// TIA Portal V16 export
// export: Created 2021-12-01T20:36:14.8298503Z, ExportSetting WithDefaults, DisplayName Totally Integrated Automation Portal, DisplayVersion V16 Update 4, DisplayName TIA Portal Version Control Interface, DisplayVersion V16 Update 2, DisplayName TIA Portal Openness, DisplayVersion V16 Update 4, DisplayName SINAMICS Startdrive Advanced, DisplayVersion V16 Update 5, DisplayName SINAMICS Startdrive G130, G150, S120, S150, SINAMICS MV, S210, DisplayVersion V16 Update 5, DisplayName SINAMICS Startdrive G110M, G120, G120C, G120D, G120P, G115D, DisplayVersion V16 Update 5, DisplayName STEP 7 Professional, DisplayVersion V16 Update 4, DisplayName STEP 7 Safety, DisplayVersion V16, DisplayName WinCC Advanced, DisplayVersion V16 Update 4
FUNCTION "ST00320_FC" : Void   // FC165, LAD
TITLE = ST00320
{ S7_Optimized_Access := 'TRUE' }
VERSION : 0.1
// stored: AutoNumber true, IsIECCheckEnabled false, SetENOAutomatically false, UDAEnableTagReadback false
   VAR_IN_OUT
      OPMODE : "OPMODE_OUT_UDT";
      HMI_EXTENSION : "HMI_EXTENSION_PANEL_UDT";
   END_VAR
   VAR_TEMP
      EmptyHS : "RT_HANDSHAKE_UDT";
   END_VAR
BEGIN

REGION Network 1: Move Opmode
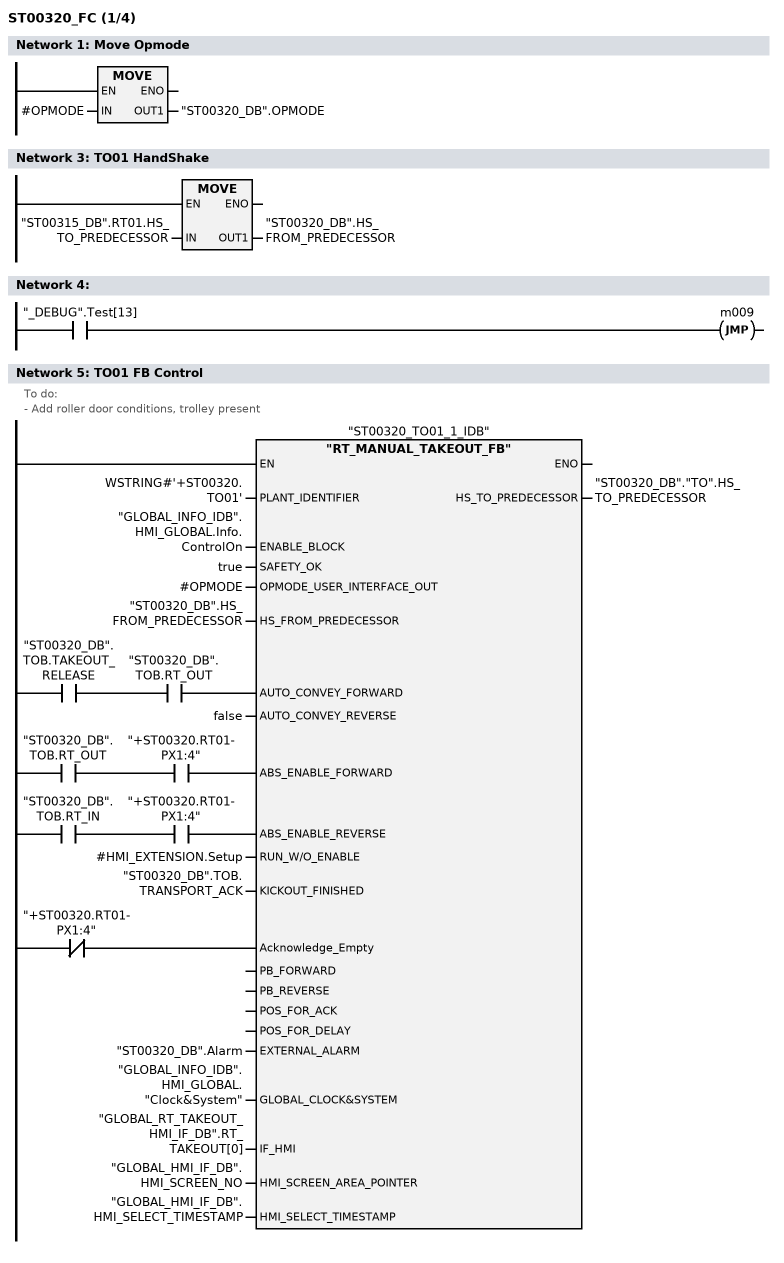
   RUNG wire#powerrail
      Move(in := #OPMODE, out1 => "ST00320_DB".OPMODE)
   END_RUNG
   // the same network as SCL:
   "ST00320_DB".OPMODE := #OPMODE;
END_REGION

REGION Network 2: *******************TO01 Control*******************
END_REGION

REGION Network 3: TO01 HandShake
   RUNG wire#powerrail
      Move(in := "ST00315_DB".RT01.HS_TO_PREDECESSOR, out1 => "ST00320_DB".HS_FROM_PREDECESSOR)
   END_RUNG
   // the same network as SCL:
   "ST00320_DB".HS_FROM_PREDECESSOR := "ST00315_DB".RT01.HS_TO_PREDECESSOR;
END_REGION

REGION Network 4
   RUNG wire#powerrail
      Contact( "_DEBUG".Test[13] )
      JumpCoil( m009 )
   END_RUNG
   // the same network as SCL:
   IF "_DEBUG".Test[13] THEN GOTO m009; END_IF;
END_REGION

REGION Network 5: TO01 FB Control
   // To do:
   // - Add roller door conditions, trolley present
   RUNG wire#powerrail
      "ST00320_TO01_1_IDB"(AUTO_CONVEY_FORWARD := wire#w1, ABS_ENABLE_FORWARD := wire#w2, ABS_ENABLE_REVERSE := wire#w3, Acknowledge_Empty := wire#w4, PLANT_IDENTIFIER := WSTRING#'+ST00320.TO01', ENABLE_BLOCK := "GLOBAL_INFO_IDB".HMI_GLOBAL.Info.ControlOn, SAFETY_OK := true, OPMODE_USER_INTERFACE_OUT := #OPMODE, HS_FROM_PREDECESSOR := "ST00320_DB".HS_FROM_PREDECESSOR, AUTO_CONVEY_REVERSE := false, "RUN_W/O_ENABLE" := #HMI_EXTENSION.Setup, KICKOUT_FINISHED := "ST00320_DB".TOB.TRANSPORT_ACK, PB_FORWARD :=, PB_REVERSE :=, POS_FOR_ACK :=, POS_FOR_DELAY :=, EXTERNAL_ALARM := "ST00320_DB".Alarm, "GLOBAL_CLOCK&SYSTEM" := "GLOBAL_INFO_IDB".HMI_GLOBAL."Clock&System", IF_HMI := "GLOBAL_RT_TAKEOUT_HMI_IF_DB".RT_TAKEOUT[0], HMI_SCREEN_AREA_POINTER := "GLOBAL_HMI_IF_DB".HMI_SCREEN_NO, HMI_SELECT_TIMESTAMP := "GLOBAL_HMI_IF_DB".HMI_SELECT_TIMESTAMP, HS_TO_PREDECESSOR => "ST00320_DB"."TO".HS_TO_PREDECESSOR)
   END_RUNG
   RUNG wire#powerrail
      Contact( "ST00320_DB".TOB.TAKEOUT_RELEASE )
      Contact( "ST00320_DB".TOB.RT_OUT )
   END_RUNG wire#w1
   RUNG wire#powerrail
      Contact( "ST00320_DB".TOB.RT_OUT )
      Contact( "+ST00320.RT01-PX1:4" )
   END_RUNG wire#w2
   RUNG wire#powerrail
      Contact( "ST00320_DB".TOB.RT_IN )
      Contact( "+ST00320.RT01-PX1:4" )
   END_RUNG wire#w3
   RUNG wire#powerrail
      I_Contact( "+ST00320.RT01-PX1:4" )
   END_RUNG wire#w4
   // the same network as SCL:
   "ST00320_TO01_1_IDB"(PLANT_IDENTIFIER := WSTRING#'+ST00320.TO01',   // "RT_MANUAL_TAKEOUT_FB"
                        ENABLE_BLOCK := "GLOBAL_INFO_IDB".HMI_GLOBAL.Info.ControlOn,
                        SAFETY_OK := true,
                        OPMODE_USER_INTERFACE_OUT := #OPMODE,
                        HS_FROM_PREDECESSOR := "ST00320_DB".HS_FROM_PREDECESSOR,
                        AUTO_CONVEY_FORWARD := "ST00320_DB".TOB.TAKEOUT_RELEASE AND "ST00320_DB".TOB.RT_OUT,
                        AUTO_CONVEY_REVERSE := false,
                        ABS_ENABLE_FORWARD := "ST00320_DB".TOB.RT_OUT AND "+ST00320.RT01-PX1:4",
                        ABS_ENABLE_REVERSE := "ST00320_DB".TOB.RT_IN AND "+ST00320.RT01-PX1:4",
                        "RUN_W/O_ENABLE" := #HMI_EXTENSION.Setup,
                        KICKOUT_FINISHED := "ST00320_DB".TOB.TRANSPORT_ACK,
                        Acknowledge_Empty := NOT "+ST00320.RT01-PX1:4",
                        EXTERNAL_ALARM := "ST00320_DB".Alarm,
                        "GLOBAL_CLOCK&SYSTEM" := "GLOBAL_INFO_IDB".HMI_GLOBAL."Clock&System",
                        IF_HMI := "GLOBAL_RT_TAKEOUT_HMI_IF_DB".RT_TAKEOUT[0],
                        HMI_SCREEN_AREA_POINTER := "GLOBAL_HMI_IF_DB".HMI_SCREEN_NO,
                        HMI_SELECT_TIMESTAMP := "GLOBAL_HMI_IF_DB".HMI_SELECT_TIMESTAMP,
                        HS_TO_PREDECESSOR => "ST00320_DB"."TO".HS_TO_PREDECESSOR);
END_REGION

REGION Network 6: Takeout Box
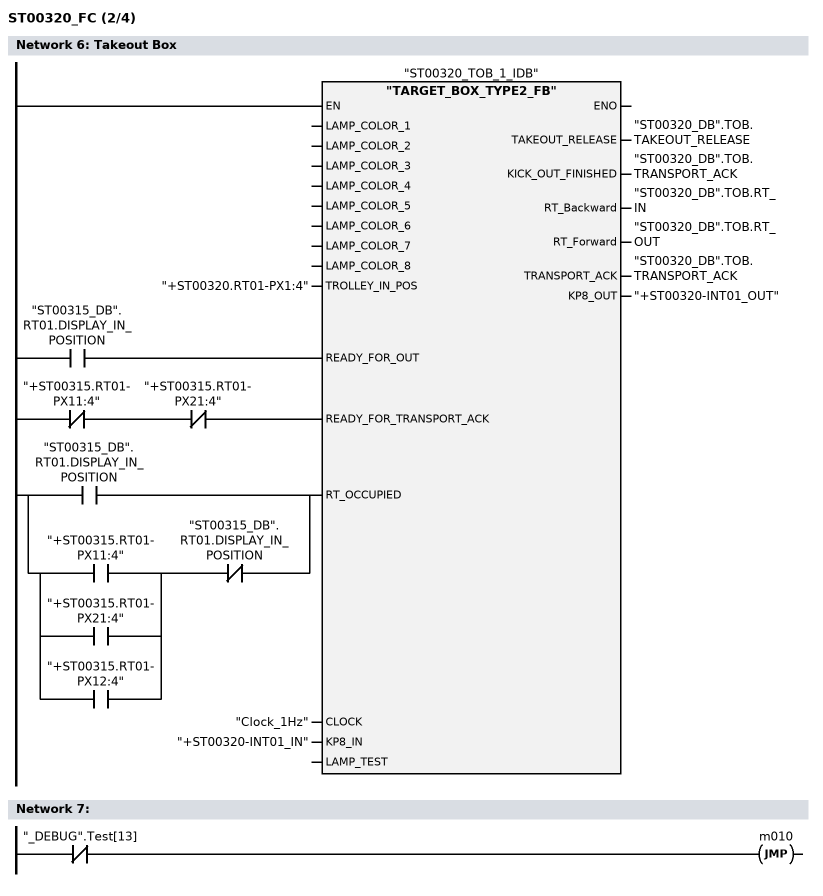
   RUNG wire#powerrail
      "ST00320_TOB_1_IDB"(READY_FOR_OUT := wire#w1, READY_FOR_TRANSPORT_ACK := wire#w2, RT_OCCUPIED := wire#w4, LAMP_COLOR_1 :=, LAMP_COLOR_2 :=, LAMP_COLOR_3 :=, LAMP_COLOR_4 :=, LAMP_COLOR_5 :=, LAMP_COLOR_6 :=, LAMP_COLOR_7 :=, LAMP_COLOR_8 :=, TROLLEY_IN_POS := "+ST00320.RT01-PX1:4", CLOCK := "Clock_1Hz", KP8_IN := "+ST00320-INT01_IN", LAMP_TEST :=, TAKEOUT_RELEASE => "ST00320_DB".TOB.TAKEOUT_RELEASE, KICK_OUT_FINISHED => "ST00320_DB".TOB.TRANSPORT_ACK, RT_Backward => "ST00320_DB".TOB.RT_IN, RT_Forward => "ST00320_DB".TOB.RT_OUT, TRANSPORT_ACK => "ST00320_DB".TOB.TRANSPORT_ACK, KP8_OUT => "+ST00320-INT01_OUT")
   END_RUNG
   RUNG wire#powerrail
      Contact( "ST00315_DB".RT01.DISPLAY_IN_POSITION )
   END_RUNG wire#w1
   RUNG wire#powerrail
      I_Contact( "+ST00315.RT01-PX11:4" )
      I_Contact( "+ST00315.RT01-PX21:4" )
   END_RUNG wire#w2
   RUNG wire#powerrail
      Contact( "ST00315_DB".RT01.DISPLAY_IN_POSITION )
   END_RUNG wire#w4
   RUNG wire#powerrail
      Contact( "+ST00315.RT01-PX11:4" )
      wire#w3
      I_Contact( "ST00315_DB".RT01.DISPLAY_IN_POSITION )
   END_RUNG wire#w4
   RUNG wire#powerrail
      Contact( "+ST00315.RT01-PX21:4" )
   END_RUNG wire#w3
   RUNG wire#powerrail
      Contact( "+ST00315.RT01-PX12:4" )
   END_RUNG wire#w3
   // the same network as SCL:
   "ST00320_TOB_1_IDB"(TROLLEY_IN_POS := "+ST00320.RT01-PX1:4",   // "TARGET_BOX_TYPE2_FB"
                       READY_FOR_OUT := "ST00315_DB".RT01.DISPLAY_IN_POSITION,
                       READY_FOR_TRANSPORT_ACK := NOT "+ST00315.RT01-PX11:4" AND NOT "+ST00315.RT01-PX21:4",
                       RT_OCCUPIED := "ST00315_DB".RT01.DISPLAY_IN_POSITION OR (("+ST00315.RT01-PX11:4" OR "+ST00315.RT01-PX21:4" OR "+ST00315.RT01-PX12:4") AND NOT "ST00315_DB".RT01.DISPLAY_IN_POSITION),
                       CLOCK := "Clock_1Hz",
                       KP8_IN := "+ST00320-INT01_IN",
                       TAKEOUT_RELEASE => "ST00320_DB".TOB.TAKEOUT_RELEASE,
                       KICK_OUT_FINISHED => "ST00320_DB".TOB.TRANSPORT_ACK,
                       RT_Backward => "ST00320_DB".TOB.RT_IN,
                       RT_Forward => "ST00320_DB".TOB.RT_OUT,
                       TRANSPORT_ACK => "ST00320_DB".TOB.TRANSPORT_ACK,
                       KP8_OUT => "+ST00320-INT01_OUT");
END_REGION

REGION Network 7
   RUNG wire#powerrail
      I_Contact( "_DEBUG".Test[13] )
      JumpCoil( m010 )
   END_RUNG
   // the same network as SCL:
   IF NOT "_DEBUG".Test[13] THEN GOTO m010; END_IF;
END_REGION

REGION Network 8: ----test----TO01 HandShake
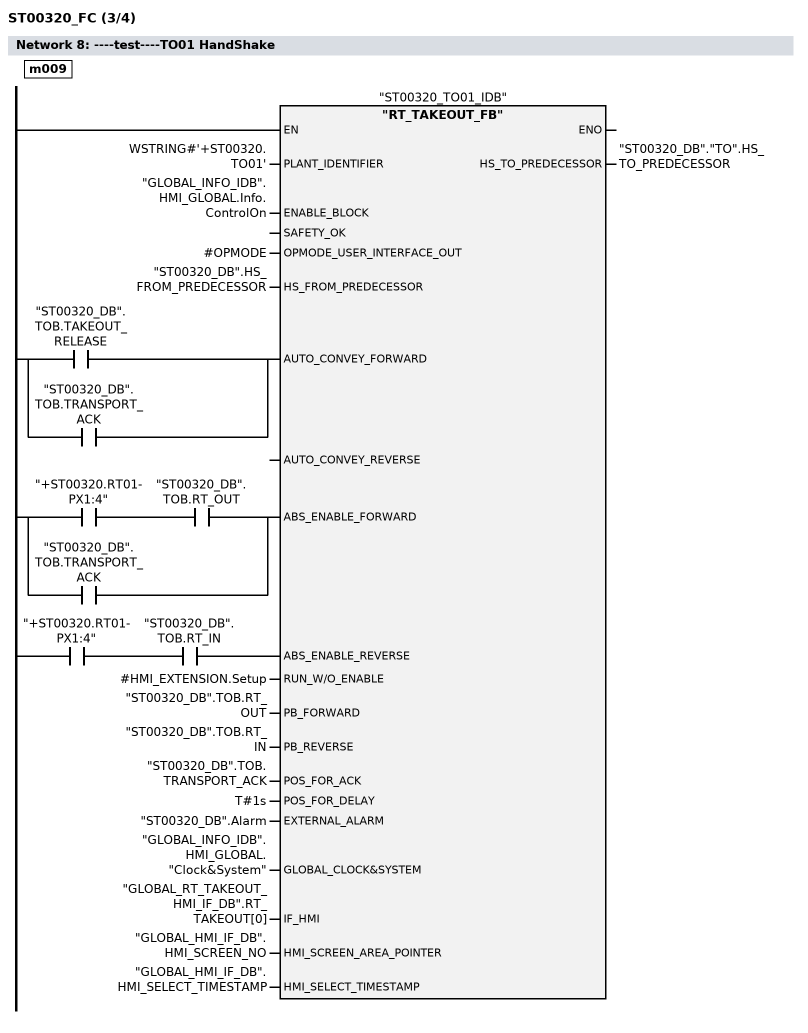
   Label( m009 )
   RUNG wire#powerrail
      "ST00320_TO01_IDB"(AUTO_CONVEY_FORWARD := wire#w1, ABS_ENABLE_FORWARD := wire#w2, ABS_ENABLE_REVERSE := wire#w3, PLANT_IDENTIFIER := WSTRING#'+ST00320.TO01', ENABLE_BLOCK := "GLOBAL_INFO_IDB".HMI_GLOBAL.Info.ControlOn, SAFETY_OK :=, OPMODE_USER_INTERFACE_OUT := #OPMODE, HS_FROM_PREDECESSOR := "ST00320_DB".HS_FROM_PREDECESSOR, AUTO_CONVEY_REVERSE :=, "RUN_W/O_ENABLE" := #HMI_EXTENSION.Setup, PB_FORWARD := "ST00320_DB".TOB.RT_OUT, PB_REVERSE := "ST00320_DB".TOB.RT_IN, POS_FOR_ACK := "ST00320_DB".TOB.TRANSPORT_ACK, POS_FOR_DELAY := T#1s, EXTERNAL_ALARM := "ST00320_DB".Alarm, "GLOBAL_CLOCK&SYSTEM" := "GLOBAL_INFO_IDB".HMI_GLOBAL."Clock&System", IF_HMI := "GLOBAL_RT_TAKEOUT_HMI_IF_DB".RT_TAKEOUT[0], HMI_SCREEN_AREA_POINTER := "GLOBAL_HMI_IF_DB".HMI_SCREEN_NO, HMI_SELECT_TIMESTAMP := "GLOBAL_HMI_IF_DB".HMI_SELECT_TIMESTAMP, HS_TO_PREDECESSOR => "ST00320_DB"."TO".HS_TO_PREDECESSOR)
   END_RUNG
   RUNG wire#powerrail
      Contact( "ST00320_DB".TOB.TAKEOUT_RELEASE )
   END_RUNG wire#w1
   RUNG wire#powerrail
      Contact( "ST00320_DB".TOB.TRANSPORT_ACK )
   END_RUNG wire#w1
   RUNG wire#powerrail
      Contact( "+ST00320.RT01-PX1:4" )
      Contact( "ST00320_DB".TOB.RT_OUT )
   END_RUNG wire#w2
   RUNG wire#powerrail
      Contact( "ST00320_DB".TOB.TRANSPORT_ACK )
   END_RUNG wire#w2
   RUNG wire#powerrail
      Contact( "+ST00320.RT01-PX1:4" )
      Contact( "ST00320_DB".TOB.RT_IN )
   END_RUNG wire#w3
   // the same network as SCL:
   m009:
   "ST00320_TO01_IDB"(PLANT_IDENTIFIER := WSTRING#'+ST00320.TO01',   // "RT_TAKEOUT_FB"
                      ENABLE_BLOCK := "GLOBAL_INFO_IDB".HMI_GLOBAL.Info.ControlOn,
                      OPMODE_USER_INTERFACE_OUT := #OPMODE,
                      HS_FROM_PREDECESSOR := "ST00320_DB".HS_FROM_PREDECESSOR,
                      AUTO_CONVEY_FORWARD := "ST00320_DB".TOB.TAKEOUT_RELEASE OR "ST00320_DB".TOB.TRANSPORT_ACK,
                      ABS_ENABLE_FORWARD := ("+ST00320.RT01-PX1:4" AND "ST00320_DB".TOB.RT_OUT) OR "ST00320_DB".TOB.TRANSPORT_ACK,
                      ABS_ENABLE_REVERSE := "+ST00320.RT01-PX1:4" AND "ST00320_DB".TOB.RT_IN,
                      "RUN_W/O_ENABLE" := #HMI_EXTENSION.Setup,
                      PB_FORWARD := "ST00320_DB".TOB.RT_OUT,
                      PB_REVERSE := "ST00320_DB".TOB.RT_IN,
                      POS_FOR_ACK := "ST00320_DB".TOB.TRANSPORT_ACK,
                      POS_FOR_DELAY := T#1s,
                      EXTERNAL_ALARM := "ST00320_DB".Alarm,
                      "GLOBAL_CLOCK&SYSTEM" := "GLOBAL_INFO_IDB".HMI_GLOBAL."Clock&System",
                      IF_HMI := "GLOBAL_RT_TAKEOUT_HMI_IF_DB".RT_TAKEOUT[0],
                      HMI_SCREEN_AREA_POINTER := "GLOBAL_HMI_IF_DB".HMI_SCREEN_NO,
                      HMI_SELECT_TIMESTAMP := "GLOBAL_HMI_IF_DB".HMI_SELECT_TIMESTAMP,
                      HS_TO_PREDECESSOR => "ST00320_DB"."TO".HS_TO_PREDECESSOR);
END_REGION

REGION Network 9: Takeout Box Standar
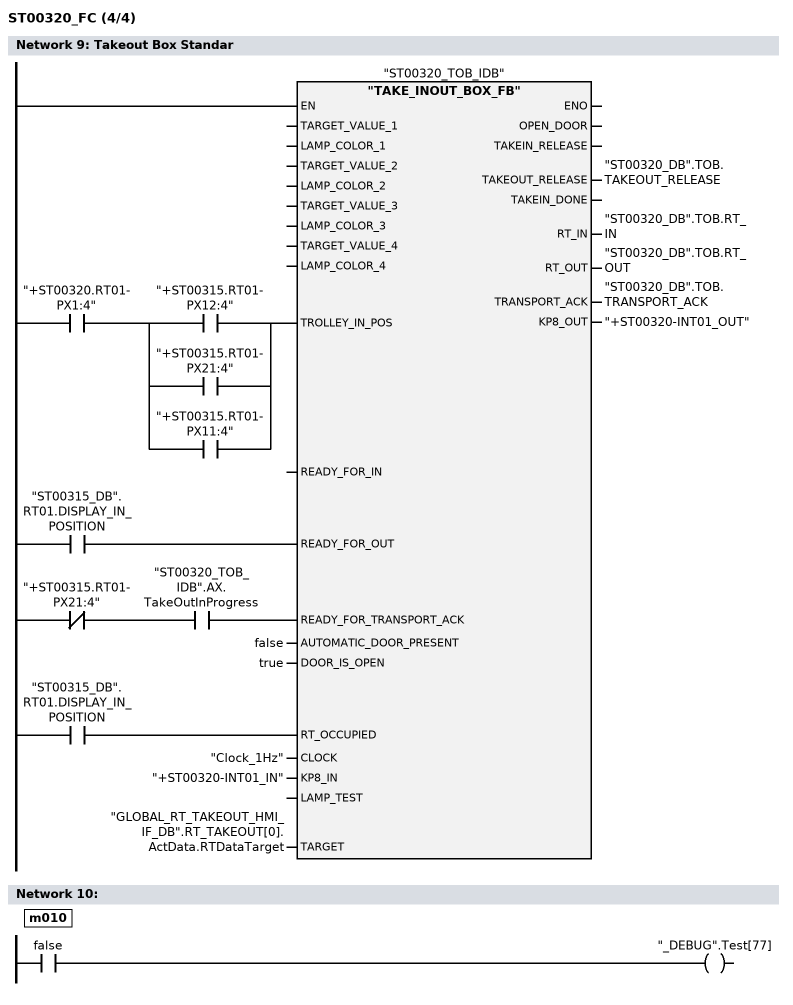
   RUNG wire#powerrail
      "ST00320_TOB_IDB"(TROLLEY_IN_POS := wire#w2, READY_FOR_OUT := wire#w3, READY_FOR_TRANSPORT_ACK := wire#w4, RT_OCCUPIED := wire#w5, TARGET_VALUE_1 :=, LAMP_COLOR_1 :=, TARGET_VALUE_2 :=, LAMP_COLOR_2 :=, TARGET_VALUE_3 :=, LAMP_COLOR_3 :=, TARGET_VALUE_4 :=, LAMP_COLOR_4 :=, READY_FOR_IN :=, AUTOMATIC_DOOR_PRESENT := false, DOOR_IS_OPEN := true, CLOCK := "Clock_1Hz", KP8_IN := "+ST00320-INT01_IN", LAMP_TEST :=, TARGET := "GLOBAL_RT_TAKEOUT_HMI_IF_DB".RT_TAKEOUT[0].ActData.RTDataTarget, OPEN_DOOR =>, TAKEIN_RELEASE =>, TAKEOUT_RELEASE => "ST00320_DB".TOB.TAKEOUT_RELEASE, TAKEIN_DONE =>, RT_IN => "ST00320_DB".TOB.RT_IN, RT_OUT => "ST00320_DB".TOB.RT_OUT, TRANSPORT_ACK => "ST00320_DB".TOB.TRANSPORT_ACK, KP8_OUT => "+ST00320-INT01_OUT")
   END_RUNG
   RUNG wire#powerrail
      Contact( "+ST00320.RT01-PX1:4" )
      wire#w1
      Contact( "+ST00315.RT01-PX12:4" )
   END_RUNG wire#w2
   RUNG wire#w1
      Contact( "+ST00315.RT01-PX21:4" )
   END_RUNG wire#w2
   RUNG wire#w1
      Contact( "+ST00315.RT01-PX11:4" )
   END_RUNG wire#w2
   RUNG wire#powerrail
      Contact( "ST00315_DB".RT01.DISPLAY_IN_POSITION )
   END_RUNG wire#w3
   RUNG wire#powerrail
      I_Contact( "+ST00315.RT01-PX21:4" )
      Contact( "ST00320_TOB_IDB".AX.TakeOutInProgress )
   END_RUNG wire#w4
   RUNG wire#powerrail
      Contact( "ST00315_DB".RT01.DISPLAY_IN_POSITION )
   END_RUNG wire#w5
   // the same network as SCL:
   "ST00320_TOB_IDB"(TROLLEY_IN_POS := "+ST00320.RT01-PX1:4" AND ("+ST00315.RT01-PX12:4" OR "+ST00315.RT01-PX21:4" OR "+ST00315.RT01-PX11:4"),   // "TAKE_INOUT_BOX_FB"
                     READY_FOR_OUT := "ST00315_DB".RT01.DISPLAY_IN_POSITION,
                     READY_FOR_TRANSPORT_ACK := NOT "+ST00315.RT01-PX21:4" AND "ST00320_TOB_IDB".AX.TakeOutInProgress,
                     AUTOMATIC_DOOR_PRESENT := false,
                     DOOR_IS_OPEN := true,
                     RT_OCCUPIED := "ST00315_DB".RT01.DISPLAY_IN_POSITION,
                     CLOCK := "Clock_1Hz",
                     KP8_IN := "+ST00320-INT01_IN",
                     TARGET := "GLOBAL_RT_TAKEOUT_HMI_IF_DB".RT_TAKEOUT[0].ActData.RTDataTarget,
                     TAKEOUT_RELEASE => "ST00320_DB".TOB.TAKEOUT_RELEASE,
                     RT_IN => "ST00320_DB".TOB.RT_IN,
                     RT_OUT => "ST00320_DB".TOB.RT_OUT,
                     TRANSPORT_ACK => "ST00320_DB".TOB.TRANSPORT_ACK,
                     KP8_OUT => "+ST00320-INT01_OUT");
END_REGION

REGION Network 10
   Label( m010 )
   RUNG wire#powerrail
      Contact( false )
      Coil( "_DEBUG".Test[77] )
   END_RUNG
   // the same network as SCL:
   m010:
   "_DEBUG".Test[77] := false;
END_REGION
END_FUNCTION
